// TIA Portal V17 export
// export: Created 2023-12-22T15:05:32.9207009Z, ExportSetting WithDefaults, DisplayName Totally Integrated Automation Portal, DisplayVersion V17, DisplayName TIA Portal Openness, DisplayVersion V17, DisplayName TIA Portal Version Control Interface, DisplayVersion V17, DisplayName STEP 7 Professional, DisplayVersion V17, DisplayName STEP 7 Safety, DisplayVersion V17, DisplayName WinCC Advanced, DisplayVersion V17
DATA_BLOCK "Time_SYS_DB"   // DB95
VERSION : 0.1
// stored: AutoNumber false, DBAccessibleFromOPCUA true, InstanceOfName Time_SYS, InstanceOfType FB
"Time_SYS"
   // VAR RETAIN
   //    Set_Time : Bool := FALSE;
   //    Time_Now : Struct
   //       Year : Int := 2020;
   //       Month : Int := 10;
   //       Day : Int := 13;
   //       Weekday : Int := 3;
   //       Hour : Int := 13;
   //       Minute : Int := 5;
   //       Second : Int := 15;
   //    END_STRUCT;
   //    Time_SP : Struct
   //       Year : Int := 2019;
   //       Month : Int := 10;
   //       Day : Int := 8;
   //       Weekday : Int := 3;
   //       Hour : Int := 14;
   //       Minute : Int := 50;
   //       Second : Int := 3;
   //    END_STRUCT;
   //    TimeZone { S7_SetPoint := 'True'} : TimeTransformationRule;
   //    RD_SYS_Status : Int := 0;
   //    WR_SYS_Status : Int := 0;
   //    RD_Time : DTL := DTL#2020-10-13-13:05:15.228830044;
   //    SP_Time : DTL := DTL#1970-01-01-00:00:00;
   //    SET_TIMEZONE { S7_SetPoint := 'True'} : SET_TIMEZONE;
   //    Time_DTL : DTL := DTL#2020-10-13-13:05:15.671240764;
   // END_VAR
BEGIN
   TimeZone.Bias := 180;
   TimeZone.DaylightBias := 60;
   TimeZone.DaylightStartMonth := 3;
   TimeZone.DaylightStartWeek := 5;
   TimeZone.DaylightStartWeekday := 7;
   TimeZone.DaylightStartHour := 2;
   TimeZone.DaylightStartMinute := 0;
   TimeZone.StandardStartMonth := 10;
   TimeZone.StandardStartWeek := 5;
   TimeZone.StandardStartWeekday := 1;
   TimeZone.StandardStartHour := 3;
   TimeZone.StandardStartMinute := 0;
   TimeZone.TimeZoneName := 'GMT+3';
   SET_TIMEZONE.REQ := FALSE;
   SET_TIMEZONE.TimeZone.Bias := 180;
   SET_TIMEZONE.TimeZone.DaylightBias := 60;
   SET_TIMEZONE.TimeZone.DaylightStartMonth := 3;
   SET_TIMEZONE.TimeZone.DaylightStartWeek := 5;
   SET_TIMEZONE.TimeZone.DaylightStartWeekday := 7;
   SET_TIMEZONE.TimeZone.DaylightStartHour := 2;
   SET_TIMEZONE.TimeZone.DaylightStartMinute := 0;
   SET_TIMEZONE.TimeZone.StandardStartMonth := 10;
   SET_TIMEZONE.TimeZone.StandardStartWeek := 5;
   SET_TIMEZONE.TimeZone.StandardStartWeekday := 1;
   SET_TIMEZONE.TimeZone.StandardStartHour := 3;
   SET_TIMEZONE.TimeZone.StandardStartMinute := 0;
   SET_TIMEZONE.TimeZone.TimeZoneName := 'GMT+3';
   SET_TIMEZONE.DONE := FALSE;
   SET_TIMEZONE.BUSY := FALSE;
   SET_TIMEZONE.ERROR := FALSE;
   SET_TIMEZONE.STATUS := 16#7000;
END_DATA_BLOCK
